# B&R Automation Studio project PallettizerProj_SM
Automation Studio 4.9

## Configuration Config1

### Task classes (Cpu.sw)
```
Cyclic#1:
  SignalHand <- SignalHandler.prg
Cyclic#2:
  Crane <- Crane.prg
  ComTCP_P <- Libraries.ComTCP.ComTCP_P.prg
  Feeder <- Feeder.prg
  InputBridg <- InputBridge.prg
  OutputBrid <- OutputBridge.prg
  PalletHand <- PalletHandler.prg
  MainContro <- MainControl.prg
Cyclic#4:
  InputFilte <- InputFilter.prg
Binaries: udbdef, FWRules, TCData, iomap, ashwac, Role, sysconf, arconfig, asfw, User, ashwd
Libraries: GenericDev, GenericAx, ComTCP_L, operator, standard, AsArLog, AsBrStr, AsTCP, SignalMng, FilterLib, asieccon, astime, runtime
```

### Hardware
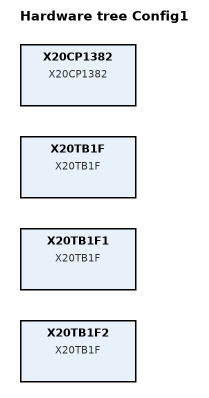
```
X20CP1382 : X20CP1382 v1.14.0.0  [X1 -> X1.SL; X2 -> X2.SL; X3 -> X3.SL]
  Module X1 (Type=X1, Virtual=true, Version=1.14.0.0)
    Connection (Connector=SS1, TargetModule=X20TB1F, TargetConnector=SS)
    Connection (Connector=SL, TargetModule=X20CP1382, TargetConnector=X1)
  Module X2 (Type=X2, Virtual=true, Version=1.14.0.0)
    Connection (Connector=SS1, TargetModule=X20TB1F1, TargetConnector=SS)
    Connection (Connector=SL, TargetModule=X20CP1382, TargetConnector=X2)
  Module X3 (Type=X3, Virtual=true, Version=1.14.0.0)
    Connection (Connector=SS1, TargetModule=X20TB1F2, TargetConnector=SS)
    Connection (Connector=SL, TargetModule=X20CP1382, TargetConnector=X3)
  Connector IF2:
    ActivateDevice = 1
  ConfigurationID = PallettizerProj2_Config1
X20TB1F : X20TB1F v1.0.0.0
X20TB1F1 : X20TB1F v1.0.0.0
X20TB1F2 : X20TB1F v1.0.0.0
```

## Configuration Default_Config

CPU 4PP065.0351-P74, AutomationRuntime C4.72, Build 4.1.2, Vc V4.72.0

### Task classes (Cpu.sw)
```
Cyclic#2:
  ComTCP_P <- Libraries.ComTCP.ComTCP_P.prg
Cyclic#4:
  InputBridg <- InputBridge.prg
  OutputBrid <- OutputBridge.prg
  MainContro <- MainControl.prg
  Feeder <- Feeder.prg
  InputFilte <- InputFilter.prg
Binaries: udbdef, mvLoader, FWRules, TCData, sysconf, Role, User, iomap, ashwd, asfw, arconfig, ashwac, TCLang
Libraries: operator, astime, standard, AsArLog, AsBrStr, AsTCP, runtime, fileio, asieccon, ComTCP_L, GenericDev, GenericAx, FilterLib
```

## Logical view

Binary libraries used (declarations not repeated): operator, runtime, astime, AsIecCon, standard, AsArLog, AsBrStr, AsTCP, MTBasics, brsystem, MTTypes, sys_lib

### Global.var - Global variables
```iecst
(*Constants*)
VAR CONSTANT
	INIT : INT := 0;
	RUN : INT := 1;
END_VAR
VAR
	START_CRANE : BOOL;
	START_PALLET_HANDLER : BOOL;
	START_MACHINE : BOOL;
	START_FEEDER : BOOL;
END_VAR
(*Insert your comment here.*)
VAR
	CraneEnabled : BOOL;
	PalletPositioned : BOOL;
	MoveCrane : BOOL;
	LayerPositioned : BOOL;
	PalletExpultion : BOOL;
	FullPalletReady : BOOL;
	PushLayer : BOOL;
	CraneHomed : BOOL;
END_VAR
(*Sensors*)
VAR
	PALLET_LIGHT_BARRIER_1_IR : BOOL;
	PALLET_LIGHT_BARRIER_2_IR : BOOL;
	LASER_SENSOR_IR : BOOL;
	VACUUM_BOX_CRANE : BOOL;
	LASER_SENSOR_2_IR : BOOL;
	pallet_light_barrier_1 : BOOL;
	pallet_light_barrier_2 : BOOL;
	laser_sensor : BOOL;
	laser_sensor2 : BOOL;
END_VAR
(*Simulation variables*)
VAR
	PUSHER_LBK : BOOL;
	PUSHER_LFR : BOOL;
	TURNPUSHER_LFR : BOOL;
	TURNPUSHER_LBK : BOOL;
	PALLET_FORK_LEFT_FB : BOOL;
	CONVEYOR_IF_FWD : BOOL;
	CONVEYOR_TURN_1_FWD : BOOL;
	PUSHER_FW : BOOL;
	CONVEYOR_END_FWD : BOOL;
	TURNPUSHER_FWD : BOOL;
	TURNPUSHER_BWD : BOOL;
	VACUUM_BOX_CRANE_GRIP : BOOL;
	CARTBOARD_TRIG : BOOL;
	SLIDE_RAIL_RIGHT_EN : BOOL;
	PUSHER_Z_EN : BOOL;
	PUSHER_X_EN : BOOL;
	PALLET_FORK_LEFT_EN : BOOL;
	PALLET_CONVEYOR_1_FWD : BOOL;
	CARRIAGE_2_AXIS : REAL;
	CARRIAGE_2_RCHD : BOOL;
	BOX_CRANE_AXIS : REAL;
	GANTRY_CRANE_AXIS : REAL;
	PALLET_LIFTER_AXIS : REAL;
	BOX_CRANE_TGT_POS : REAL;
	CARRIAGE_2_TGT_POS : REAL;
	GANTRY_CRANE_TGT_POS : REAL;
	PALLET_LIFTER_TGT_POS : REAL;
	PALLET_CONVEYOR_2_ACT_VEL : REAL;
END_VAR
(*Variables*)
VAR
	OperationType : INT := 0;
END_VAR
```

### MNG_Package.var
```iecst
(*                                                                            *)
(* File generated by the B&R AS 4 control config generator                    *)
(*                                                                            *)
(*     Provider: machineering                                                 *)
(*  Application: industrialPhysics_2.4.master                                 *)
(* Architecture: Windows 64 Bit                                               *)
(*      Version: 2.4.10491.master                                             *)
(*        Build: 164f85bec                                                    *)
(*         Date: 2020-05-19, Time: 12:11:21                                   *)
(*                                                                            *)
VAR
	ComTCP_SimInputs : ComTCP_INPUTS_32BIT := (0);
	ComTCP_SimOutputs : ComTCP_OUTPUTS_32BIT := (0);
	ComTCP_SimServerAddress : STRING[15] := '127.0.0.1';
	ComTCP_SimServerPort : UINT := 5000;
	ComTCP_SimSendCycleTime : TIME := T#5ms;
	ComTCP_SimActive : BOOL := FALSE;
END_VAR
(*Signal for the SignalMng*)
VAR
	OnPhaseStopHMI : BOOL;
	AuxReset : BOOL;
	Reset : BOOL;
	ImmediateStopHMI : BOOL;
	NoMorePallet : BOOL;
	OnPhaseStop : BOOL;
	ImmediateStop : BOOL;
	EmergencyStop : BOOL;
	ConveyorIfFault : BOOL;
	ConveyorIfFaultHMI : BOOL;
	ConveyorTurnFault : BOOL;
	ConveyorTurnFaultHMI : BOOL;
	TurnPusherFault : BOOL;
	TurnPusherFaultHMI : BOOL;
	PusherFault : BOOL;
	PusherFaultHMI : BOOL;
	ConveyorEndFault : BOOL;
	ConveyorEndFaultHMI : BOOL;
	CarriageFault : BOOL;
	CarriageFaultHMI : BOOL;
END_VAR
```

### Package Logical/Libraries - Global libraries

### Library Logical/Libraries/GenericDev (IEC)

#### GenericDevice.st
```iecst
(* TODO: Add your comment here *)
FUNCTION_BLOCK GenericDevice

	// Device Clock Handler

	IF (DeviceClock AND (DeviceTimer > 0))THEN
		DeviceTimer := DeviceTimer - 1;
	END_IF;

	// Device Initialization handler

	CASE (DeviceType AND DEVICE_FEEDBACK_MASK) OF

		DEVICE_WITH_ENABLE_FEEDBACK:
			DeviceDisabledSensor := NOT DeviceEnabledSensor AND
			((DeviceState = DeviceDisabledState) OR (DeviceState = DeviceDisablePhaseState AND DeviceTimeout));

			DeviceDisabled := NOT DeviceEnabled AND
			((DeviceState = DeviceDisabledState) OR
			(DeviceState = DeviceDisablePhaseState AND DeviceTimeout));

		DEVICE_WITH_DISABLE_FEEDBACK :
			DeviceEnabled := NOT DeviceDisabled AND
			((DeviceState = DeviceEnabledState) OR
			(DeviceState = DeviceEnablePhaseState AND DeviceTimeout));

			DeviceEnabledSensor := NOT DeviceDisabledSensor AND
			((DeviceState = DeviceEnabledState) OR (DeviceState = DeviceEnablePhaseState AND DeviceTimeout));

		DEVICE_WITHOUT_FEEDBACK:
			DeviceEnabled := (DeviceState = DeviceEnabledState) OR
			(DeviceState = DeviceEnablePhaseState AND DeviceTimeout);
			DeviceDisabled := (DeviceState = DeviceDisabledState) OR
			(DeviceState = DeviceDisablePhaseState AND DeviceTimeout);

			DeviceEnabledSensor := (DeviceState = DeviceEnabledState) OR ((DeviceState = DeviceEnablePhaseState) AND DeviceTimeout);
			DeviceDisabledSensor := (DeviceState = DeviceDisabledState) OR ((DeviceState = DeviceDisablePhaseState) AND DeviceTimeout);
	END_CASE;

	IF (DeviceOperation = INIT) THEN
		// Device sensor handler
		CASE (DeviceType AND DEVICE_FEEDBACK_MASK) OF

			DEVICE_WITH_ENABLE_FEEDBACK:
				DeviceDisabled := NOT DeviceEnabled;

			DEVICE_WITH_DISABLE_FEEDBACK :
				DeviceEnabled := NOT DeviceDisabled;

			DEVICE_WITHOUT_FEEDBACK:
				DeviceEnabled := DeviceEnablePreset;
				DeviceDisabled := NOT DeviceEnabled;
		END_CASE;

		DeviceEnableRequest := FALSE;
		DeviceDisableRequest := FALSE;
		IF (DeviceEnablePreset) THEN
			EnableDevice := TRUE;
			DeviceTimer := DeviceEnableTime;
			IF (NOT (DeviceDisabled AND DeviceEnabled)) THEN
				DeviceState := DeviceEnablePhaseState;
			ELSE
				DeviceState := DeviceEnabledState;
			END_IF;
			DeviceNotInitialized := NOT DeviceEnabled OR DeviceDisabled;
		ELSE
			EnableDevice := FALSE;
			DeviceTimer := DeviceDisableTime;
			IF (NOT (DeviceDisabled AND DeviceEnabled)) THEN
				DeviceState := DeviceDisablePhaseState;
			ELSE
				DeviceState := DeviceDisabledState;
			END_IF;
			DeviceNotInitialized := (DeviceEnabled OR NOT DeviceDisabled);
		END_IF;
	END_IF;

	//	Device control handler

	CASE (DeviceState) OF

		DeviceDisabledState:
			DeviceDisableRequest := FALSE;
			IF (DeviceEnableRequest) THEN
				EnableDevice := TRUE;
				DeviceTimer := DeviceEnableTime;
				DeviceState := DeviceEnablePhaseState;
			END_IF;

		DeviceEnablePhaseState:
			IF DeviceDisableRequest THEN
				DeviceEnableRequest	:= FALSE;
				EnableDevice	:= FALSE;
				DeviceTimer	:= DeviceDisableTime;
				DeviceState	:= DeviceDisablePhaseState;
			END_IF;
			IF DeviceEnabledSensor THEN
				DeviceEnableRequest := FALSE;
				DeviceTimer	:= 0;
				DeviceState := DeviceEnabledState;
			END_IF;

		DeviceEnabledState:
			DeviceEnableRequest	:= FALSE;
			IF DeviceDisableRequest THEN
				EnableDevice := FALSE;
				DeviceTimer	:= DeviceDisableTime;
				DeviceState := DeviceDisablePhaseState;
			END_IF;

		DeviceDisablePhaseState:
			IF DeviceEnableRequest THEN
				DeviceDisableRequest	:= FALSE;
				EnableDevice	:= TRUE;
				DeviceTimer	:= DeviceEnableTime;
				DeviceState	:= DeviceEnablePhaseState;
			END_IF;

			IF DeviceDisabledSensor THEN
				DeviceDisableRequest := FALSE;
				DeviceTimer	:= 0;
				DeviceState := DeviceDisabledState;
			END_IF;

	END_CASE;

	// Device Diagnostic handler

	DeviceTimeout := (DeviceTimer = 0);

	DeviceDisabledSensorFault := ( NOT EnableDevice AND NOT DeviceDisabledSensor AND NOT DeviceEnabledSensor OR EnableDevice AND DeviceDisabledSensor AND DeviceEnabledSensor) AND DeviceTimeout;

	DeviceEnabledSensorFault := (NOT EnableDevice AND DeviceDisabledSensor AND DeviceEnabledSensor OR EnableDevice AND NOT DeviceDisabledSensor AND NOT DeviceEnabledSensor) AND DeviceTimeout;

	DeviceActuatorFault := (NOT EnableDevice AND NOT DeviceDisabledSensor AND DeviceEnabledSensor OR EnableDevice AND DeviceDisabledSensor AND NOT DeviceEnabledSensor) AND DeviceTimeout;

	DeviceFault :=	DeviceDisabledSensorFault OR DeviceEnabledSensorFault OR DeviceActuatorFault;

	// Device actuators handler

	CASE (DeviceType AND DEVICE_ACTUATION_MASK) OF

		DEVICE_WITH_DOUBLE_ACTUATION:
			DisableDevice := NOT EnableDevice;

		DEVICE_WITH_DA_NO_RETAIN:
			EnableDevice := EnableDevice AND (DeviceState = DeviceEnablePhaseState);
			DisableDevice := NOT EnableDevice AND (DeviceState = DeviceDisablePhaseState);

	END_CASE;

END_FUNCTION_BLOCK
```

### Library Logical/Libraries/GenericAx (IEC)

#### Constants.var
```iecst
VAR CONSTANT
	IDLE : WORD := 0;
	CHANGE_VELOCITY : WORD := 1;
	CHANGE_POSITION : WORD := 2;
	IMMEDIATE_STOP_REQUEST : WORD := 3;
	EMERGENCY_STOP_REQUEST : WORD := 4;
END_VAR
```

#### GenericAx.fun
```iecst
FUNCTION_BLOCK GenericAxis
	VAR_INPUT
		Command : WORD := 0;
		ActualPosition : REAL;
		ActualVelocity : REAL;
		NewSetPoint : REAL;
		DeviceTimer : INT;
		TGT_SENSOR : BOOL;
		Reset : BOOL;
	END_VAR
	VAR_OUTPUT
		TargetVelocity : REAL;
		TargetPosition : REAL;
		InPosition : BOOL := 1;
		InVelocity : BOOL := 1;
		DeviceFault : BOOL;
		AxisBusy : BOOL;
	END_VAR
	VAR
		AxisState : GA_State := CheckCommand;
		Timer : INT;
	END_VAR
END_FUNCTION_BLOCK
```

#### GenericAxis.st
```iecst
(* TODO: Add your comment here *)
FUNCTION_BLOCK GenericAxis

	CASE (AxisState) OF

		CheckCommand:

			//			IF Command = IDLE THEN
			//				Timer	:= DeviceTimer;
			//				DeviceFault	:= FALSE;
			//			END_IF;

			IF Command = CHANGE_POSITION THEN

				IF (ActualPosition <> NewSetPoint) THEN
					Timer	:= DeviceTimer;
					InPosition	:= FALSE;
					TargetPosition := NewSetPoint;
					AxisState := WaitTargetPosition;
				END_IF

			END_IF;

			IF Command = CHANGE_VELOCITY THEN

				IF (ActualVelocity <> NewSetPoint) THEN
					Timer	:= DeviceTimer;
					TargetVelocity := NewSetPoint;
					InVelocity	:= FALSE;
					AxisState	:= WaitTargetVelocity;
				END_IF

			END_IF;

//			IF Command = IMMEDIATE_STOP_REQUEST THEN
//
//				TargetPosition	:= ActualPosition;
//				TargetVelocity	:= 0;
//				IF (ActualPosition = TargetPosition AND ActualVelocity = TargetVelocity) THEN
//					InPosition	:= TRUE;
//					InVelocity	:= TRUE;
//					AxisState	:= CheckCommand;
//				END_IF;
//
//			END_IF;

			IF Command = EMERGENCY_STOP_REQUEST THEN
				TargetPosition	:= ActualPosition;
				TargetVelocity	:= 0;
				IF (ActualPosition = TargetPosition AND ActualVelocity = TargetVelocity) THEN
					InPosition	:= TRUE;
					InVelocity	:= TRUE;
					AxisState	:= CheckCommand;
				END_IF;
			END_IF;

		WaitTargetPosition:
			IF (ActualPosition = TargetPosition AND TGT_SENSOR) THEN
				InPosition	:= TRUE;
				AxisState	:= CheckCommand;
			END_IF;
			Timer	:= Timer	- 1;
			IF Timer = 0 THEN
				DeviceFault	:= TRUE;
				AxisState	:= FaultState;
			END_IF;

		WaitTargetVelocity:
			IF ActualVelocity = TargetVelocity THEN
				InVelocity	:= TRUE;
				AxisState	:= CheckCommand;
			END_IF;
			Timer	:= Timer	- 1;
			IF Timer = 0 THEN
				DeviceFault	:= TRUE;
				AxisState	:= FaultState;
			END_IF;

		FaultState:
			IF Reset THEN
				DeviceFault	:= FALSE;
				AxisState	:= CheckCommand;
			END_IF;

	END_CASE;

END_FUNCTION_BLOCK
```

### Library Logical/Libraries/SignalMng (IEC)

#### SignalManagement.st
```iecst
(* TODO: Add your comment here *)
FUNCTION_BLOCK SignalManagement

	CASE SignalOperation OF

		START_CONFIGURATION: (* reset signal count*)

			NumberOfAlarms := 0;
			NumberOfAnomalies := 0;
			NumberOfInformation := 0;
			NumberOfWarnings := 0;

		CONFIGURATION:

			CASE (SignalType AND SIGNAL_TYPE_MASK) OF
				ALARM:
					NumberOfAlarms := NumberOfAlarms + 1;
				ANOMALY:
					NumberOfAnomalies := NumberOfAnomalies + 1;
				WARNING:
					NumberOfWarnings := NumberOfWarnings + 1;
				INFORMATION:
					NumberOfInformation := NumberOfInformation + 1;
			END_CASE

		START_GENERATION:

			ResetEnable := FALSE;
			SignalOutputs := NONE;
			ResetActivation := Reset AND NOT ResetOld;
			ResetOld := Reset;
			AuxResetEnable	:= FALSE;
			AuxResetActivation := KeyReset AND NOT KeyResetOld;
			KeyResetOld:= KeyReset;

		GENERATION:
			CASE (SignalType AND SIGNAL_TYPE_MASK) OF
				ALARM:
					Index := NumberOfActiveAlarms;
					BaseIndex := 0;
					Condition := TRUE;
				ANOMALY:
					Index := NumberOfActiveAnomalies;
					BaseIndex := NumberOfAlarms;
					Condition := TRUE;
				WARNING:
					Index := NumberOfActiveWarning;
					BaseIndex := NumberOfAlarms + NumberOfAnomalies;
					Condition := TRUE;
				INFORMATION:
					Index := NumberOfActiveInformation;
					BaseIndex := NumberOfAlarms + NumberOfAnomalies + NumberOfWarnings;
					Condition := TRUE;
			END_CASE

			IF ActivationSignal AND NOT Signals[SignalCode] THEN
				Signals[SignalCode] := TRUE;
				Index := Index + 1;
				ActiveSignalCodes[BaseIndex + Index] := SignalCode;
			END_IF

			AuxResetRequired := ((SignalType AND AUX_RESET) = AUX_RESET);

			IF (Condition AND Signals[SignalCode] AND NOT ActivationSignal AND (ActiveSignalCodes[BaseIndex + 1] = SignalCode) AND AuxResetRequired) THEN
				AuxResetEnable := TRUE; // LED AUX RECOVERY GREEN
			END_IF

			IF (Condition AND Signals[SignalCode] AND NOT ActivationSignal AND (ActiveSignalCodes[BaseIndex + 1] = SignalCode)) THEN
				ResetEnable := TRUE; // LED RECOVERY GREEN
			END_IF

			IF ((ResetActivation OR NOT Condition) AND Signals[SignalCode] AND NOT ActivationSignal AND (ActiveSignalCodes[BaseIndex + 1] = SignalCode)) THEN
				Signals[SignalCode] := FALSE;

				FOR i := 2 TO Index DO
					ActiveSignalCodes[BaseIndex + i-1] := ActiveSignalCodes[BaseIndex + i];
				END_FOR;

				ActiveSignalCodes[BaseIndex + Index] := 0;
				Index := Index - 1;
				ResetActivation := FALSE;
			END_IF

			IF ((AuxResetActivation OR NOT Condition) AND Signals[SignalCode] AND NOT ActivationSignal AND (ActiveSignalCodes[BaseIndex + 1] = SignalCode) AND AuxResetRequired) THEN
				Signals[SignalCode] := FALSE;

				FOR i := 2 TO Index DO
					ActiveSignalCodes[BaseIndex + i-1] := ActiveSignalCodes[BaseIndex + i];
				END_FOR;

				ActiveSignalCodes[BaseIndex + Index] := 0;
				Index := Index - 1;
				AuxResetActivation := FALSE;
			END_IF

			CASE (SignalType AND SIGNAL_TYPE_MASK) OF
				ALARM:
					NumberOfActiveAlarms := Index;
				ANOMALY:
					NumberOfActiveAnomalies := Index;
				WARNING:
					NumberOfActiveWarning := Index;
				INFORMATION:
					NumberOfActiveInformation := Index;
			END_CASE

			IF Signals[SignalCode] THEN
				SignalOutputs := SignalOutputs OR SignalOutput;
			END_IF

		RUN_SM:
			CurrentAlarm := NumberOfActiveAlarms;
			CurrentAnomaly := NumberOfActiveAnomalies;
			CurrentWarning := NumberOfActiveWarning;
			CurrentInformation := NumberOfActiveInformation;

			IF NumberOfActiveAlarms > 0 THEN
				ActiveAlarmCode := ActiveSignalCodes[CurrentAlarm];
			ELSE
				ActiveAlarmCode := SignalCodeDefault;
			END_IF

			IF NumberOfActiveAnomalies > 0 THEN
				ActiveAnomalyCode := ActiveSignalCodes[NumberOfAlarms + CurrentAnomaly];
			ELSE
				ActiveAnomalyCode := SignalCodeDefault;
			END_IF

			IF NumberOfActiveWarning > 0 THEN
				ActiveWarningCode := ActiveSignalCodes[NumberOfAlarms + NumberOfAnomalies + CurrentWarning];
			ELSE
				ActiveWarningCode := SignalCodeDefault;
			END_IF

			IF NumberOfActiveInformation > 0 THEN
				ActiveInformationCode := ActiveSignalCodes[NumberOfAlarms + NumberOfAnomalies + NumberOfWarnings + CurrentInformation];
			ELSE
				ActiveInformationCode := SignalCodeDefault;
			END_IF;

	END_CASE

END_FUNCTION_BLOCK
```

### Library Logical/Libraries/FilterLib (IEC)

#### FilterLib.fun - Exported functions and function blocks
```iecst
(**)

{REDUND_ERROR} FUNCTION_BLOCK MyFilterFB (*TODO: Add your comment here*) (*$GROUP=User,$CAT=User,$GROUPICON=User.png,$CATICON=User.png*)
	VAR_INPUT
		OperationType : INT;
		Clock : BOOL;
		Signal : BOOL;
		ActivationDelay : UDINT;
		DeactivationDelay : UDINT;
	END_VAR
	VAR_OUTPUT
		DelayedSignal : BOOL;
	END_VAR
	VAR
		Delay : UDINT;
	END_VAR
END_FUNCTION_BLOCK
```

#### MyFilterFB.st
```iecst
(* TODO: Add your comment here *)
FUNCTION_BLOCK MyFilterFB
	IF (OperationType = 0) THEN
		Delay := 0;
	END_IF;
	IF (Clock AND (Delay > 0)) THEN
		Delay := Delay - 1;
	END_IF;
	IF (Delay = 0) THEN
		DelayedSignal := Signal;
	END_IF;
	IF (Signal = DelayedSignal)	THEN
		IF (Signal) THEN
			Delay := DeactivationDelay;
		ELSE
			Delay := ActivationDelay;

		END_IF;
	END_IF;
END_FUNCTION_BLOCK
```

### Program Logical/MainControl (IEC)

#### Main.st
```iecst
PROGRAM _INIT
	(* Insert code here *)

END_PROGRAM

PROGRAM _CYCLIC

	CASE MainState OF

		Initialization:

			IF (OperationType = INIT) THEN

				OperationType := RUN;
				MainState := WaitStart;

			END_IF

		WaitStart:

			IF(START_MACHINE) THEN

				START_FEEDER := TRUE;
				START_CRANE := TRUE;
				START_PALLET_HANDLER := TRUE;
				MainState := WaitCrane;
			END_IF

		WaitCrane:

			IF CraneHomed THEN

				PushLayer := TRUE;
				MainState := WaitFeeder;

			END_IF

			IF FullPalletReady THEN

				PalletExpultion := TRUE;
				MainState := WaitPalletHandler;

			END_IF

		WaitFeeder:

			IF LayerPositioned THEN

				MoveCrane := TRUE;
				MainState := WaitPalletHandler;

			END_IF

		WaitPalletHandler:

			IF OnPhaseStop AND PalletExpultion THEN
				MainState := StopMachine;
			END_IF

			IF PalletPositioned AND NOT (OnPhaseStop AND PalletExpultion) THEN

				CraneEnabled := TRUE;
				MainState := WaitCrane;

			END_IF

		StopMachine:

			START_MACHINE := FALSE;
			START_FEEDER := FALSE;
			START_CRANE := FALSE;
			START_PALLET_HANDLER := FALSE;

			IF Reset THEN

				MainState := WaitStart;

			END_IF

	END_CASE

END_PROGRAM

PROGRAM _EXIT
	(* Insert code here *)

END_PROGRAM
```

### Program Logical/Feeder (IEC)

#### Types.typ
```iecst
TYPE
	FeederStateType :
		(
		WaitStart,
		WaitConv,
		PusherBox,
		BoxCounting,
		BackwardCarriage,
		WaitingBack,
		WaitSyncCrane,
		StopFeederImmediate,
		StopFeederOnPhase,
		WaitingForReactivation
		);
	FeederStruct : 	STRUCT
		State : FeederStateType;
		Start : BOOL;
		Conveyor_if : GenericDevice;
		Conveyor_if_enable_request : BOOL;
		Conveyor_if_disable_request : BOOL;
		Conveyor_if_EnableTime : INT := 20;
		Conveyor_if_DisableTime : INT := 20;
		Conveyor_turn1 : GenericDevice;
		Conveyor_turn1_disable_request : BOOL;
		Conveyor_turn1_enable_request : BOOL;
		Conveyor_turn1_EnableTime : INT := 20;
		Conveyor_turn1_DisableTime : INT := 20;
		Pusher : GenericDevice;
		Pusher_disable_request : BOOL;
		Pusher_enable_request : BOOL;
		PusherEnableTime : INT := 200;
		PusherDisableTime : INT := 200;
		Conveyor_end : GenericDevice;
		Conveyor_end_disable_request : BOOL;
		Conveyor_end_enable_request : BOOL;
		Conveyor_end_EnableTime : INT := 20;
		Conveyor_end_DisableTime : INT := 20;
		Turnpusher : GenericDevice;
		Turnpusher_enable_request : BOOL;
		Turnpusher_disable_request : BOOL;
		TurnpusherEnableTime : INT := 200;
		TurnpusherDisableTime : INT := 200;
		Carriage : GenericAxis;
		CarriagePositionReached : BOOL;
	END_STRUCT;
END_TYPE
```

#### Variables.var
```iecst
VAR
	StopRequest : BOOL := FALSE;
	Box : INT;
	Format : INT := 1;
	Line : INT := 1;
	F_TRIG_0 : F_TRIG;
	LaserSensor2 : BOOL;
	LayerOn : BOOL;
	Feeder : FeederStruct;
	LastLayer : BOOL;
	PrevState : FeederStateType;
	ExpectedBox : INT;
END_VAR
```

#### Main.st
```iecst
PROGRAM _INIT
	(* Insert code here *)

END_PROGRAM

PROGRAM _CYCLIC

	// Falling edge in the coining boxes sensor
	F_TRIG_0( CLK:=LASER_SENSOR_2_IR );
	LaserSensor2 := F_TRIG_0.Q;

	Feeder.Start := START_FEEDER;

	CASE (Feeder.State) OF

		WaitStart:

			IF ImmediateStop THEN

				PrevState := WaitStart;
				Feeder.State := StopFeederImmediate;

			ELSIF Feeder.Start THEN

				Feeder.Conveyor_if_enable_request := TRUE;
				Feeder.Conveyor_turn1_enable_request := TRUE;
				Feeder.Conveyor_end_enable_request := TRUE;

				Feeder.State := WaitConv;

			END_IF

		WaitConv:

			IF ImmediateStop THEN

				Feeder.Conveyor_if_disable_request := TRUE;
				Feeder.Conveyor_end_disable_request := TRUE;
				Feeder.Conveyor_turn1_disable_request := TRUE;

				PrevState := WaitConv;
				Feeder.State := StopFeederImmediate;

			ELSIF NOT Feeder.Conveyor_if_enable_request AND NOT Feeder.Conveyor_turn1_enable_request AND NOT Feeder.Conveyor_end_enable_request THEN

				Feeder.State := PusherBox;

			END_IF

		PusherBox:

			IF ImmediateStop THEN

				Feeder.Conveyor_if_disable_request := TRUE;
				Feeder.Conveyor_end_disable_request := TRUE;
				Feeder.Conveyor_turn1_disable_request := TRUE;

				PrevState := PusherBox;
				Feeder.State := StopFeederImmediate;

			// Behaviour with an OnPhase stop signal
			ELSIF LastLayer AND OnPhaseStop THEN

				Feeder.Conveyor_if_disable_request := TRUE;
				Feeder.Conveyor_end_disable_request := TRUE;
				Feeder.State := StopFeederOnPhase;

			// Nominal behaviour
			ELSIF NOT Feeder.Turnpusher_enable_request AND NOT Feeder.Turnpusher_disable_request AND Feeder.CarriagePositionReached THEN

				IF LASER_SENSOR_IR AND NOT Feeder.Pusher_disable_request THEN
					ExpectedBox := Box + 1;
					Feeder.Pusher_enable_request := TRUE;
					LastLayer := FALSE;
					Feeder.State := BoxCounting;
				END_IF

				IF Box <> ExpectedBox THEN
					Feeder.Pusher_enable_request := TRUE;
					LastLayer := FALSE;
					Feeder.State := BoxCounting;
				END_IF

			END_IF

		BoxCounting:

			IF ImmediateStop THEN

				Feeder.Conveyor_if_disable_request := TRUE;
				Feeder.Conveyor_end_disable_request := TRUE;
				Feeder.Conveyor_turn1_disable_request := TRUE;
				PrevState := BoxCounting;
				Feeder.State := StopFeederImmediate;

			// Nominal
			ELSIF NOT Feeder.Pusher_enable_request THEN

				Feeder.Pusher_disable_request := TRUE;
				LayerPositioned := FALSE;
				LayerOn := FALSE;

				IF LaserSensor2 THEN
					Box := Box+1;

					// Type of boxes in the pallet (first horizzontals)
					IF Format = 1 AND Line = 1 AND Box = 8 THEN
						Feeder.Turnpusher_enable_request := TRUE;
						Line := 2;
						Box := 0;
						ExpectedBox := 0;
						Feeder.Carriage.NewSetPoint	:= 0.44;
						Feeder.Carriage.Command := CHANGE_POSITION;
						Feeder.State := BackwardCarriage;
					END_IF

					IF Format = 1 AND Line = 2 AND Box = 3 THEN
						Line := 3;
						Feeder.Carriage.NewSetPoint	:= 0.44;
						Feeder.Carriage.Command := CHANGE_POSITION;
						Feeder.State := BackwardCarriage;
					END_IF

					IF Format = 1 AND Line = 3 AND Box = 6 THEN
						Line := 1;
						Format := 2;
						Box := 0;
						ExpectedBox := 0;
						Feeder.State := WaitSyncCrane;
					END_IF

					IF Format = 2 AND Line = 1 AND Box = 3 THEN
						Line := 2;
						Feeder.Carriage.NewSetPoint	:= 0.44;
						Feeder.Carriage.Command := CHANGE_POSITION;
						Feeder.State := BackwardCarriage;
					END_IF

					IF Format = 2 AND Line = 2 AND Box = 6 THEN
						Feeder.Turnpusher_disable_request := TRUE;
						Line := 3;
						Box := 0;
						ExpectedBox := 0;
						Feeder.Carriage.NewSetPoint := 0.44;
						Feeder.Carriage.Command := CHANGE_POSITION;
						Feeder.State := BackwardCarriage;
					END_IF

					IF Format = 2 AND Line = 3 AND Box = 8 THEN
						LastLayer := TRUE;
						Line := 1;
						Format := 1;
						Box := 0;
						ExpectedBox := 0;
						Feeder.State := WaitSyncCrane;
					END_IF

					IF (Feeder.State <> BackwardCarriage) AND (Feeder.State <> WaitSyncCrane) THEN
						Feeder.State := PusherBox;
					END_IF
				END_IF

			END_IF

		BackwardCarriage:

			IF ImmediateStop THEN

				Feeder.Conveyor_if_disable_request := TRUE;
				Feeder.Conveyor_end_disable_request := TRUE;
				Feeder.Conveyor_turn1_disable_request := TRUE;

				PrevState := BackwardCarriage;
				Feeder.State := StopFeederImmediate;

			ELSIF Feeder.CarriagePositionReached THEN

				Feeder.Carriage.NewSetPoint := 0.0;
				Feeder.Carriage.Command := CHANGE_POSITION;
				Feeder.State := WaitingBack;

			END_IF

		WaitingBack:

			IF ImmediateStop THEN

				Feeder.Conveyor_if_disable_request := TRUE;
				Feeder.Conveyor_end_disable_request := TRUE;
				Feeder.Conveyor_turn1_disable_request := TRUE;

				PrevState := WaitingBack;
				Feeder.State := StopFeederImmediate;

			ELSIF LayerOn AND Feeder.CarriagePositionReached THEN
				LayerPositioned := TRUE;
				Feeder.State := PusherBox;

			ELSIF NOT LayerOn AND Feeder.CarriagePositionReached THEN
				Feeder.State := PusherBox;
			END_IF

		WaitSyncCrane:

			IF ImmediateStop THEN

				Feeder.Conveyor_if_disable_request := TRUE;
				Feeder.Conveyor_end_disable_request := TRUE;
				Feeder.Conveyor_turn1_disable_request := TRUE;

				PrevState := WaitSyncCrane;
				Feeder.State := StopFeederImmediate;

			ELSIF PushLayer THEN
				Feeder.Carriage.NewSetPoint	:= 1.1;
				Feeder.Carriage.Command := CHANGE_POSITION;
				LayerOn := TRUE;
				PushLayer := FALSE;
				Feeder.State := BackwardCarriage;
			END_IF

		StopFeederImmediate:

			IF LaserSensor2 THEN
				Box := Box+1;
			END_IF

			IF  NOT Feeder.Conveyor_if_disable_request AND NOT Feeder.Conveyor_end_disable_request AND NOT Feeder.Conveyor_turn1_disable_request
				AND NOT ImmediateStop THEN

				Feeder.Conveyor_if_enable_request := TRUE;
				Feeder.Conveyor_end_enable_request := TRUE;
				Feeder.Conveyor_turn1_enable_request := TRUE;
				Feeder.State := WaitingForReactivation;

			END_IF

		StopFeederOnPhase:

			IF NOT Feeder.Conveyor_if_disable_request AND NOT Feeder.Conveyor_end_disable_request AND NOT OnPhaseStop AND NOT ImmediateStop THEN

				Feeder.State := WaitStart;

			END_IF

		WaitingForReactivation:

			IF LaserSensor2 THEN
				Box := Box+1;
			END_IF

			IF NOT Feeder.Conveyor_if_enable_request AND NOT Feeder.Conveyor_end_enable_request AND NOT Feeder.Conveyor_turn1_enable_request THEN

				IF Box <> ExpectedBox THEN
					Feeder.State := BoxCounting;
				END_IF

				IF Box = ExpectedBox THEN
					Feeder.Pusher_disable_request := TRUE;
					Feeder.State := PusherBox;
				END_IF

			END_IF

	END_CASE

	Feeder.Conveyor_if.DeviceOperation := OperationType;
	Feeder.Conveyor_if.DeviceClock := TRUE;
	Feeder.Conveyor_if.DeviceDiagnosticsEnabled := TRUE;
	Feeder.Conveyor_if.DeviceEnablePreset := FALSE;
	Feeder.Conveyor_if.DeviceEnableTime := Feeder.Conveyor_if_EnableTime;
	Feeder.Conveyor_if.DeviceDisableTime := Feeder.Conveyor_if_DisableTime;
	Feeder.Conveyor_if.DeviceType := DEVICE_WITHOUT_FEEDBACK OR DEVICE_WITH_SINGLE_ACTUATION;
	Feeder.Conveyor_if(DeviceEnableRequest := Feeder.Conveyor_if_enable_request, DeviceDisableRequest := Feeder.Conveyor_if_disable_request);
	CONVEYOR_IF_FWD := Feeder.Conveyor_if.EnableDevice;
	ConveyorIfFault	:= Feeder.Conveyor_if.DeviceFault;

	Feeder.Conveyor_turn1.DeviceOperation := OperationType;
	Feeder.Conveyor_turn1.DeviceClock := TRUE;
	Feeder.Conveyor_turn1.DeviceDiagnosticsEnabled := TRUE;
	Feeder.Conveyor_turn1.DeviceEnablePreset := FALSE;
	Feeder.Conveyor_turn1.DeviceEnableTime := Feeder.Conveyor_turn1_EnableTime;
	Feeder.Conveyor_turn1.DeviceDisableTime := Feeder.Conveyor_turn1_DisableTime;
	Feeder.Conveyor_turn1.DeviceType := DEVICE_WITHOUT_FEEDBACK OR DEVICE_WITH_SINGLE_ACTUATION;
	Feeder.Conveyor_turn1(DeviceEnableRequest := Feeder.Conveyor_turn1_enable_request, DeviceDisableRequest := Feeder.Conveyor_turn1_disable_request);
	CONVEYOR_TURN_1_FWD := Feeder.Conveyor_turn1.EnableDevice;
	ConveyorTurnFault := Feeder.Conveyor_turn1.DeviceFault;

	Feeder.Pusher.DeviceOperation := OperationType;
	Feeder.Pusher.DeviceClock := TRUE;
	Feeder.Pusher.DeviceDiagnosticsEnabled := TRUE;
	Feeder.Pusher.DeviceEnablePreset := FALSE;
	Feeder.Pusher.DeviceEnabledSensor := PUSHER_LFR;
	Feeder.Pusher.DeviceDisabledSensor := PUSHER_LBK;
	Feeder.Pusher.DeviceEnableTime := Feeder.PusherEnableTime;
	Feeder.Pusher.DeviceDisableTime := Feeder.PusherDisableTime;
	Feeder.Pusher.DeviceType := DEVICE_WITH_DOUBLE_FEEDBACK OR DEVICE_WITH_SINGLE_ACTUATION;
	Feeder.Pusher(DeviceEnableRequest := Feeder.Pusher_enable_request, DeviceDisableRequest := Feeder.Pusher_disable_request);
	PUSHER_FW := Feeder.Pusher.EnableDevice;
	PusherFault := Feeder.Pusher.DeviceActuatorFault;

	Feeder.Conveyor_end.DeviceOperation := OperationType;
	Feeder.Conveyor_end.DeviceClock := TRUE;
	Feeder.Conveyor_end.DeviceDiagnosticsEnabled := TRUE;
	Feeder.Conveyor_end.DeviceEnablePreset := FALSE;
	Feeder.Conveyor_end.DeviceEnableTime := Feeder.Conveyor_end_EnableTime;
	Feeder.Conveyor_end.DeviceDisableTime := Feeder.Conveyor_end_DisableTime;
	Feeder.Conveyor_end.DeviceType := DEVICE_WITHOUT_FEEDBACK OR DEVICE_WITH_SINGLE_ACTUATION;
	Feeder.Conveyor_end(DeviceEnableRequest := Feeder.Conveyor_end_enable_request, DeviceDisableRequest := Feeder.Conveyor_end_disable_request);
	CONVEYOR_END_FWD := Feeder.Conveyor_end.EnableDevice;
	ConveyorEndFault:= Feeder.Conveyor_end.DeviceFault;

	Feeder.Turnpusher.DeviceOperation := OperationType;
	Feeder.Turnpusher.DeviceClock := TRUE;
	Feeder.Turnpusher.DeviceDiagnosticsEnabled := TRUE;
	Feeder.Turnpusher.DeviceEnablePreset := FALSE;
	Feeder.Turnpusher.DeviceEnabledSensor := TURNPUSHER_LBK;
	Feeder.Turnpusher.DeviceDisabledSensor := TURNPUSHER_LFR;
	Feeder.Turnpusher.DeviceEnableTime := Feeder.TurnpusherEnableTime;
	Feeder.Turnpusher.DeviceDisableTime := Feeder.TurnpusherDisableTime;
	Feeder.Turnpusher.DeviceType := DEVICE_WITH_DOUBLE_FEEDBACK OR DEVICE_WITH_DOUBLE_ACTUATION;
	Feeder.Turnpusher(DeviceEnableRequest := Feeder.Turnpusher_enable_request, DeviceDisableRequest := Feeder.Turnpusher_disable_request);
	TURNPUSHER_BWD := Feeder.Turnpusher.EnableDevice;
	TURNPUSHER_FWD := Feeder.Turnpusher.DisableDevice;
	TurnPusherFault := Feeder.Turnpusher.DeviceActuatorFault;

	Feeder.Carriage.ActualPosition	:= CARRIAGE_2_AXIS;
	CARRIAGE_2_TGT_POS	:= Feeder.Carriage.TargetPosition;
	Feeder.Carriage.TGT_SENSOR	:= CARRIAGE_2_RCHD;
	Feeder.Carriage.DeviceTimer := 400;
	CarriageFault := Feeder.Carriage.DeviceFault;
	Feeder.Carriage();
	Feeder.CarriagePositionReached	:= Feeder.Carriage.InPosition;

END_PROGRAM

PROGRAM _EXIT
	(* Insert code here *)

END_PROGRAM
```

### Program Logical/Crane (IEC)

#### Variables.var
```iecst
VAR
	Crane : CraneStruct;
	NextLayer : INT := 1;
	PrevState : CraneStateType := GoBack;
	CraneState : CraneStateType := 0;
	BoxCraneAxisBusy : BOOL;
	NextState : CraneStateType;
	CompleatingPallet : BOOL;
END_VAR
```

#### Main.st
```iecst
PROGRAM _INIT
	(* Insert code here *)

END_PROGRAM

PROGRAM _CYCLIC

	Crane.Start := START_CRANE;

	CASE (Crane.State) OF

		WaitStart:
			IF Crane.Start THEN
				Crane.State := MoveCraneForCartboard;
			END_IF

		WaitLayer:
			IF Crane.BoxCranePositionReached THEN
				CraneHomed := TRUE;

				IF MoveCrane THEN
					MoveCrane := FALSE;
					Crane.PusherZ_enable_request := TRUE;
					Crane.SlideRail_enable_request := TRUE;
					CraneHomed := FALSE;
					IF (NextLayer = 1) THEN
						Crane.State := ReleaseFirstCartboard;
					END_IF

					IF (NextLayer = 2) THEN
						Crane.State := ReleaseSecondCartboard;
					END_IF
				END_IF
			END_IF

		ReleaseFirstCartboard:

			IF (NOT Crane.PusherZ_enable_request AND NOT Crane.SlideRail_enable_request) AND CraneEnabled THEN

				NextLayer := 2;
				PrevState := ReleaseFirstCartboard;
				Crane.GantryCrane.NewSetPoint := -1.11;
				Crane.GantryCrane.Command := CHANGE_POSITION;
				Crane.BoxCrane.NewSetPoint := -0.2;
				Crane.BoxCrane.Command := CHANGE_POSITION;
				Crane.State := WaitingPositioning;

			END_IF

		PositioningLayer:

			IF NOT Crane.Vacuum_disable_request AND NOT VACUUM_BOX_CRANE THEN

				PrevState := PositioningLayer;
				Crane.GantryCrane.NewSetPoint := -1.3;
				Crane.GantryCrane.Command := CHANGE_POSITION;
				Crane.State := WaitingPositioning;

			END_IF

		LayerOnPallet:

			IF NOT Crane.SlideRail_disable_request THEN

				Crane.PusherX_enable_request := TRUE ;
				Crane.GantryCrane.NewSetPoint := 0.0;
				Crane.GantryCrane.Command := CHANGE_POSITION;
				PrevState := LayerOnPallet;
				Crane.State := WaitingPositioning;

			END_IF

		GoBack:

			IF FullPalletReady AND OnPhaseStop THEN

				Crane.PusherZ_disable_request := TRUE;
				Crane.PusherX_disable_request := TRUE;
				Crane.BoxCrane.NewSetPoint := 0.0;
				Crane.BoxCrane.Command := CHANGE_POSITION;
				NextState := StopCrane;
				PrevState := GoBack;
				Crane.State := WaitingPositioning;

			END_IF

			CraneEnabled := FALSE;
			FullPalletReady := FALSE;

			IF PrevState = LayerOnPallet AND NOT Crane.PusherX_enable_request THEN

				Crane.PusherZ_disable_request := TRUE;
				Crane.PusherX_disable_request := TRUE;
				Crane.BoxCrane.NewSetPoint := 0.0;
				Crane.BoxCrane.Command := CHANGE_POSITION;
				NextState := MoveCraneForCartboard;
				PrevState := GoBack;
				Crane.State := WaitingPositioning;

			END_IF

			IF (PrevState = LoadCartboard AND NOT Crane.Vacuum_enable_request) THEN

				Crane.BoxCrane.NewSetPoint := 0.0;
				Crane.BoxCrane.Command := CHANGE_POSITION;
				NextState := WaitLayer;
				PrevState := GoBack;
				Crane.State := WaitingPositioning;

			END_IF

		MoveCraneForCartboard:

			IF Crane.BoxCranePositionReached THEN

				Crane.BoxCrane.NewSetPoint := -0.195;
				Crane.BoxCrane.Command := CHANGE_POSITION;
				Crane.State := LoadCartboard;

			END_IF

		LoadCartboard:

			IF Crane.BoxCranePositionReached THEN

				Crane.Vacuum_enable_request	:= TRUE;
				Crane.Cartboard_enable_request := TRUE;
				PrevState := LoadCartboard;
				Crane.State := GoBack;

			END_IF

		ReleaseSecondCartboard:

			IF (NOT Crane.PusherZ_enable_request AND NOT Crane.SlideRail_enable_request) THEN

				NextLayer := 1;
				Crane.GantryCrane.NewSetPoint := -1.11;
				Crane.GantryCrane.Command := CHANGE_POSITION;
				Crane.BoxCrane.NewSetPoint := 0.01;
				Crane.BoxCrane.Command := CHANGE_POSITION;
				CompleatingPallet := TRUE;
				PrevState := ReleaseSecondCartboard;
				Crane.State := WaitingPositioning;

			END_IF

		WaitingPositioning:

			IF Crane.GantryCranePositionReached AND Crane.BoxCranePositionReached    (*GANTRY_CRANE_AXIS = -1.11 AND BOX_CRANE_AXIS = 0.01*) THEN

				IF PrevState = ReleaseFirstCartboard OR PrevState = ReleaseSecondCartboard THEN

					Crane.Vacuum_disable_request := TRUE;
					Crane.Cartboard_disable_request := TRUE;
					Crane.State := PositioningLayer;

				END_IF

				IF PrevState = PositioningLayer THEN

					Crane.SlideRail_disable_request := TRUE;
					Crane.State := LayerOnPallet;

				END_IF

				IF PrevState = LayerOnPallet THEN

					IF CompleatingPallet THEN
						CompleatingPallet:=FALSE;
						FullPalletReady := TRUE;
					END_IF

					Crane.State := GoBack;

				END_IF

				IF PrevState = GoBack THEN

					Crane.State := NextState;

				END_IF

			END_IF

		StopCrane:

			IF Reset THEN

				Crane.State := WaitStart;

			END_IF

	END_CASE

	Crane.Vacuum.DeviceOperation := OperationType;
	Crane.Vacuum.DeviceClock := TRUE;
	Crane.Vacuum.DeviceDiagnosticsEnabled := TRUE;
	Crane.Vacuum.DeviceEnablePreset := FALSE;
	Crane.Vacuum.DeviceEnabledSensor := VACUUM_BOX_CRANE;
	Crane.Vacuum.DeviceEnableTime := 500;//VacuumEnableTime;
	Crane.Vacuum.DeviceDisableTime := Crane.VacuumDisableTime;
	Crane.Vacuum.DeviceType := DEVICE_WITH_SINGLE_ACTUATION OR DEVICE_WITH_ENABLE_FEEDBACK;
	Crane.Vacuum(DeviceEnableRequest := Crane.Vacuum_enable_request, DeviceDisableRequest := Crane.Vacuum_disable_request );
	VACUUM_BOX_CRANE_GRIP := Crane.Vacuum.EnableDevice;
	//eVacuumFault := (*Vacuum.DeviceEnabledSensorFault OR Vacuum.DeviceActuatorFault*) SIMVacuumFault;

	Crane.Cartboard.DeviceOperation := OperationType;
	Crane.Cartboard.DeviceClock := TRUE;
	Crane.Cartboard.DeviceDiagnosticsEnabled := TRUE;
	Crane.Cartboard.DeviceEnablePreset := FALSE;
	Crane.Cartboard.DeviceEnableTime := Crane.CartboardEnableTime;
	Crane.Cartboard.DeviceDisableTime := Crane.CartboardDisableTime;
	Crane.Cartboard.DeviceType := DEVICE_WITHOUT_FEEDBACK OR DEVICE_WITH_SINGLE_ACTUATION;
	Crane.Cartboard(DeviceEnableRequest := Crane.Cartboard_enable_request, DeviceDisableRequest := Crane.Cartboard_disable_request);
	CARTBOARD_TRIG := Crane.Cartboard.EnableDevice;
//	eCartboardFault	:= (*Cartboard.DeviceActuatorFault*) SIMCartboardFault;

	Crane.SlideRail.DeviceOperation := OperationType;
	Crane.SlideRail.DeviceClock := TRUE;
	Crane.SlideRail.DeviceDiagnosticsEnabled := TRUE;
	Crane.SlideRail.DeviceEnablePreset := FALSE;
	Crane.SlideRail.DeviceEnableTime := Crane.SlideRailEnableTime;
	Crane.SlideRail.DeviceDisableTime := Crane.SlideRailDisableTime;
	Crane.SlideRail.DeviceType := DEVICE_WITHOUT_FEEDBACK OR DEVICE_WITH_SINGLE_ACTUATION;
	Crane.SlideRail(DeviceEnableRequest := Crane.SlideRail_enable_request, DeviceDisableRequest := Crane.SlideRail_disable_request);
	SLIDE_RAIL_RIGHT_EN := Crane.SlideRail.EnableDevice;
	//eSlideRailFault	:= (*SlideRail.DeviceActuatorFault*) SIMSlideRailFault;

	Crane.PusherZ.DeviceOperation := OperationType;
	Crane.PusherZ.DeviceClock := TRUE;
	Crane.PusherZ.DeviceDiagnosticsEnabled := TRUE;
	Crane.PusherZ.DeviceEnablePreset := FALSE;
	Crane.PusherZ.DeviceEnableTime := Crane.PusherZEnableTime;
	Crane.PusherZ.DeviceDisableTime := Crane.PusherZDisableTime;
	Crane.PusherZ.DeviceType := DEVICE_WITHOUT_FEEDBACK OR DEVICE_WITH_SINGLE_ACTUATION;
	Crane.PusherZ(DeviceEnableRequest := Crane.PusherZ_enable_request, DeviceDisableRequest := Crane.PusherZ_disable_request);
	PUSHER_Z_EN := Crane.PusherZ.EnableDevice;
	//ePusherzFault	:= (*PusherZ.DeviceActuatorFault*) SIMPusherzFault;

	Crane.PusherX.DeviceOperation := OperationType;
	Crane.PusherX.DeviceClock := TRUE;
	Crane.PusherX.DeviceDiagnosticsEnabled := TRUE;
	Crane.PusherX.DeviceEnablePreset := FALSE;
	Crane.PusherX.DeviceEnableTime := Crane.PusherXEnableTime;
	Crane.PusherX.DeviceDisableTime := Crane.PusherXDisableTime;
	Crane.PusherX.DeviceType := DEVICE_WITHOUT_FEEDBACK OR DEVICE_WITH_SINGLE_ACTUATION;
	Crane.PusherX(DeviceEnableRequest := Crane.PusherX_enable_request, DeviceDisableRequest := Crane.PusherX_disable_request );
	PUSHER_X_EN := Crane.PusherX.EnableDevice;
	//ePusherxFault	:= (*PusherX.DeviceActuatorFault*) SIMPusherxFault;

	Crane.GantryCrane.ActualPosition	:= GANTRY_CRANE_AXIS;
	Crane.GantryCrane.TGT_SENSOR	:= TRUE;
	GANTRY_CRANE_TGT_POS	:= Crane.GantryCrane.TargetPosition;
	Crane.GantryCrane.DeviceTimer	:= 400;
	//eGantryCraneFault	:= (*GantryCrane.DeviceFault*) SIMGantryCraneFault;
	Crane.GantryCrane();
	Crane.GantryCranePositionReached	:= Crane.GantryCrane.InPosition;

	//BoxCrane.NewSetPoint	:= BoxCraneSetPoint;
	Crane.BoxCrane.ActualPosition	:= BOX_CRANE_AXIS;
	Crane.BoxCrane.TGT_SENSOR	:= TRUE;
	BOX_CRANE_TGT_POS	:=	Crane.BoxCrane.TargetPosition;
	Crane.BoxCrane.DeviceTimer	:= 400;
	//eBoxCraneFault	:= (*BoxCrane.DeviceFault*) SIMBoxCraneFault;
	Crane.BoxCrane();
	Crane.BoxCranePositionReached	:= Crane.BoxCrane.InPosition;

END_PROGRAM

PROGRAM _EXIT
	(* Insert code here *)

END_PROGRAM
```

### Program Logical/PalletHandler (IEC)

#### Types.typ
```iecst
TYPE
	PalletStruct : 	STRUCT
		Start : BOOL;
		State : PalletStateType;
		PalletFork : GenericDevice;
		PalletFork_enable_request : BOOL;
		PalletFork_disable_request : BOOL;
		PalletForkEnableTime : INT := 20;
		PalletForkDisableTime : INT := 20;
		PalletLifter : GenericAxis;
		PalletLifterPositionReached : BOOL;
		PalletConveyor1 : GenericDevice;
		PalletConveyor1EnableTime : INT := 20;
		PalletConveyor1DisableTime : INT := 20;
		PalletConveyor2 : GenericAxis;
		PalletConveyor1_disable_request : BOOL;
		PalletConveyor1_enable_request : BOOL;
		PalletConveyor2VelocityReached : BOOL;
	END_STRUCT;
	PalletStateType :
		(
		WaitStart,
		ReleasePallet,
		NextPallet,
		LifterHoming,
		MovingPallet,
		PositioningPallet,
		PalletApproaching,
		PalletInPosition,
		WaitingPositioning,
		StopPalletOnPhase,
		StopPalletImmediate
		);
END_TYPE
```

#### Main.st
```iecst
PROGRAM _INIT

	NumberPallet := 5;

END_PROGRAM

PROGRAM _CYCLIC

	Pallet.Start := START_PALLET_HANDLER;

	CASE (Pallet.State) OF

		WaitStart:

			IF ImmediateStop THEN

				PrevState := WaitStart;
				Pallet.State := StopPalletImmediate;

			ELSIF Pallet.Start THEN
				Pallet.State := ReleasePallet;
			END_IF

		ReleasePallet:

			PalletExpultion := FALSE;
			PalletPositioned := FALSE;

			IF ImmediateStop THEN

				Pallet.PalletConveyor2.NewSetPoint := 0.0;
				Pallet.PalletConveyor2.Command := CHANGE_VELOCITY;

				PrevState := ReleasePallet;
				Pallet.State :=StopPalletImmediate;

			ELSIF Pallet.PalletLifterPositionReached AND NOT OnPhaseStop THEN

				Pallet.PalletConveyor2.NewSetPoint := 0.5;
				Pallet.PalletConveyor2.Command := CHANGE_VELOCITY;
				Pallet.PalletLifter.NewSetPoint := -0.258;
				Pallet.PalletLifter.Command := CHANGE_POSITION;

				PrevState := ReleasePallet;
				Pallet.State := WaitingPositioning;

			END_IF

		NextPallet:

			IF ImmediateStop THEN

				Pallet.PalletConveyor2.NewSetPoint := 0.0;
				Pallet.PalletConveyor2.Command := CHANGE_VELOCITY;

				PrevState := NextPallet;
				Pallet.State :=StopPalletImmediate;

			ELSIF NOT Pallet.PalletFork_enable_request THEN

				Pallet.PalletLifter.NewSetPoint := -0.12;
				Pallet.PalletLifter.Command := CHANGE_POSITION;

				PrevState := NextPallet;
				Pallet.State := WaitingPositioning;

			END_IF

		LifterHoming:

			IF ImmediateStop THEN

				Pallet.PalletConveyor2.NewSetPoint := 0.0;
				Pallet.PalletConveyor2.Command := CHANGE_VELOCITY;

				PrevState := LifterHoming;
				Pallet.State :=StopPalletImmediate;

			ELSIF NOT Pallet.PalletFork_disable_request THEN
				Pallet.PalletLifter.NewSetPoint := 0.0;
				Pallet.PalletLifter.Command := CHANGE_POSITION;

				Pallet.State := MovingPallet;
			END_IF

		MovingPallet:

			IF ImmediateStop THEN

				Pallet.PalletConveyor2.NewSetPoint := 0.0;
				Pallet.PalletConveyor2.Command := CHANGE_VELOCITY;

				PrevState := MovingPallet;
				Pallet.State :=StopPalletImmediate;

			ELSIF Pallet.PalletLifterPositionReached THEN

				Pallet.PalletConveyor1_enable_request := TRUE;
				Pallet.PalletLifter.NewSetPoint := 0.0;
				Pallet.PalletLifter.Command := CHANGE_POSITION;
				Pallet.State := PositioningPallet;

			END_IF

		PositioningPallet:

			IF ImmediateStop THEN

				Pallet.PalletConveyor2.NewSetPoint := 0.0;
				Pallet.PalletConveyor2.Command := CHANGE_VELOCITY;
				Pallet.PalletConveyor1_disable_request := TRUE;

				PrevState := PositioningPallet;
				Pallet.State :=StopPalletImmediate;

			ELSIF Pallet.PalletConveyor2VelocityReached AND NOT Pallet.PalletConveyor1_enable_request AND PALLET_LIGHT_BARRIER_2_IR THEN

				Pallet.PalletConveyor2.NewSetPoint := 0.1;
				Pallet.PalletConveyor2.Command := CHANGE_VELOCITY;
				Pallet.State := PalletApproaching;

			END_IF

		PalletApproaching:

			IF ImmediateStop THEN

				Pallet.PalletConveyor2.NewSetPoint := 0.0;
				Pallet.PalletConveyor2.Command := CHANGE_VELOCITY;
				Pallet.PalletConveyor1_disable_request := TRUE;

				PrevState := PalletApproaching;
				Pallet.State :=StopPalletImmediate;

			ELSIF Pallet.PalletConveyor2VelocityReached AND PALLET_LIGHT_BARRIER_1_IR THEN

				Pallet.PalletConveyor2.NewSetPoint := 0.0;
				Pallet.PalletConveyor2.Command := CHANGE_VELOCITY;
				Pallet.PalletConveyor1_disable_request := TRUE;
				Pallet.State := PalletInPosition;

			END_IF

		PalletInPosition:

			IF ImmediateStop THEN

				PrevState := PalletApproaching;
				Pallet.State :=StopPalletImmediate;

			ELSIF Pallet.PalletConveyor2VelocityReached AND NOT Pallet.PalletConveyor1_disable_request THEN

				PalletPositioned := TRUE;

				IF PalletExpultion THEN

					IF OnPhaseStop THEN

						Pallet.PalletConveyor1_disable_request := TRUE;
						Pallet.PalletConveyor2.NewSetPoint := 0.0;
						Pallet.PalletConveyor2.Command := CHANGE_VELOCITY;
						Pallet.State := StopPalletOnPhase;

					END_IF

					IF NOT OnPhaseStop THEN

						Pallet.PalletConveyor2.NewSetPoint := 0.5;
						Pallet.PalletConveyor2.Command := CHANGE_VELOCITY;
						Pallet.State := ReleasePallet;

					END_IF

				END_IF

			END_IF

		WaitingPositioning:

			IF ImmediateStop THEN

				Pallet.PalletConveyor2.NewSetPoint := 0.0;
				Pallet.PalletConveyor2.Command := CHANGE_VELOCITY;
				Pallet.State := StopPalletImmediate;

			ELSIF Pallet.PalletLifterPositionReached THEN

				IF PrevState = ReleasePallet THEN
					NumberPallet := NumberPallet-1;

					IF NumberPallet = 0 THEN
						NoMorePallet := TRUE;
					END_IF

					Pallet.PalletFork_enable_request := TRUE;
					Pallet.State := NextPallet;

				END_IF

				IF PrevState = NextPallet THEN

					Pallet.PalletFork_disable_request := TRUE;
					Pallet.State := LifterHoming;

				END_IF

			END_IF

		StopPalletOnPhase:

			IF NOT Pallet.PalletConveyor1_disable_request AND Pallet.PalletConveyor2VelocityReached  AND NOT OnPhaseStop THEN

				IF NumberPallet = 0 THEN
					NoMorePallet := FALSE;
					NumberPallet := 5;
				END_IF

				Pallet.State := WaitStart;

			END_IF

		StopPalletImmediate:

			IF Pallet.PalletConveyor2VelocityReached AND NOT ImmediateStop THEN

				IF (PrevState = PositioningPallet ) AND NOT Pallet.PalletConveyor1_disable_request THEN

					Pallet.PalletConveyor1_enable_request := TRUE;
					Pallet.PalletConveyor2.NewSetPoint := 0.5;
					Pallet.PalletConveyor2.Command := CHANGE_VELOCITY;

				END_IF

				IF PrevState = PalletApproaching AND NOT Pallet.PalletConveyor1_disable_request THEN

					Pallet.PalletConveyor1_enable_request := TRUE;
					Pallet.PalletConveyor2.NewSetPoint := 0.1;
					Pallet.PalletConveyor2.Command := CHANGE_VELOCITY;

				END_IF

				Pallet.State := PrevState;

			END_IF

	END_CASE

	Pallet.PalletFork.DeviceOperation := OperationType;
	Pallet.PalletFork.DeviceClock := TRUE;
	Pallet.PalletFork.DeviceDiagnosticsEnabled := TRUE;
	Pallet.PalletFork.DeviceEnablePreset := FALSE;
	Pallet.PalletFork.DeviceEnabledSensor := PALLET_FORK_LEFT_FB;
	Pallet.PalletFork.DeviceEnableTime := Pallet.PalletForkEnableTime;
	Pallet.PalletFork.DeviceDisableTime := Pallet.PalletForkDisableTime;
	PALLET_FORK_LEFT_EN := Pallet.PalletFork.EnableDevice;
	Pallet.PalletFork.DeviceType := DEVICE_WITH_ENABLE_FEEDBACK OR DEVICE_WITH_SINGLE_ACTUATION;
	Pallet.PalletFork(DeviceEnableRequest := Pallet.PalletFork_enable_request, DeviceDisableRequest := Pallet.PalletFork_disable_request);
	PalletforkFault := Pallet.PalletFork.DeviceFault;

	Pallet.PalletConveyor1.DeviceOperation := OperationType;
	Pallet.PalletConveyor1.DeviceClock := TRUE;
	Pallet.PalletConveyor1.DeviceDiagnosticsEnabled := TRUE;
	Pallet.PalletConveyor1.DeviceEnablePreset := FALSE;
	Pallet.PalletConveyor1.DeviceEnableTime := Pallet.PalletConveyor1EnableTime;
	Pallet.PalletConveyor1.DeviceDisableTime := Pallet.PalletConveyor1DisableTime;
	Pallet.PalletConveyor1.DeviceType := DEVICE_WITHOUT_FEEDBACK OR DEVICE_WITH_SINGLE_ACTUATION;
	PALLET_CONVEYOR_1_FWD := Pallet.PalletConveyor1.EnableDevice;
	Pallet.PalletConveyor1(DeviceEnableRequest := Pallet.PalletConveyor1_enable_request, DeviceDisableRequest := Pallet.PalletConveyor1_disable_request);
	PalletConveyor1Fault := Pallet.PalletConveyor1.DeviceFault;

	Pallet.PalletLifter.ActualPosition	:= PALLET_LIFTER_AXIS;
	Pallet.PalletLifter.TGT_SENSOR	:= TRUE;
	PALLET_LIFTER_TGT_POS 	:= Pallet.PalletLifter.TargetPosition;
	Pallet.PalletLifter.DeviceTimer	:= 400;
	PalletLifterFault	:= Pallet.PalletLifter.DeviceFault;
	Pallet.PalletLifter();
	Pallet.PalletLifterPositionReached	:= Pallet.PalletLifter.InPosition;

	Pallet.PalletConveyor2.ActualVelocity	:= PALLET_CONVEYOR_2_ACT_VEL;
	PALLET_CONVEYOR_2_ACT_VEL	:= Pallet.PalletConveyor2.TargetVelocity;
	Pallet.PalletConveyor2.DeviceTimer	:= 400;
	PalletConveyor2Fault:= Pallet.PalletConveyor2.DeviceFault;
	Pallet.PalletConveyor2();
	Pallet.PalletConveyor2VelocityReached	:= Pallet.PalletConveyor2.InVelocity;

END_PROGRAM

PROGRAM _EXIT
	(* Insert code here *)

END_PROGRAM
```

### Program Logical/SignalHandler (IEC)

#### Main.st
```iecst
PROGRAM _INIT
	(* Insert code here *)

END_PROGRAM

PROGRAM _CYCLIC

	// Recognize input

	IF (OperationType = INIT) THEN
		SignalManager(SignalOperation := START_CONFIGURATION);
		SignalManager.SignalOperation  := CONFIGURATION;
	ELSE
		SignalManager(SignalOperation 	:= START_GENERATION);
		SignalManager.SignalOperation 	:= GENERATION;
	END_IF;

	SignalManager.ActivationSignal := OnPhaseStopHMI;
	SignalManager.SignalCode := 1;
	SignalManager.SignalType := ANOMALY;
	SignalManager.SignalOutput := ON_PHASE_STOP;
	SignalManager.Reset := Reset;
	SignalManager();

	SignalManager.ActivationSignal := NoMorePallet;
	SignalManager.SignalCode := 2;
	SignalManager.SignalType := ANOMALY;
	SignalManager.SignalOutput := ON_PHASE_STOP;
	SignalManager.Reset := Reset;
	SignalManager();

	SignalManager.ActivationSignal := ImmediateStopHMI;
	SignalManager.SignalCode := 3;
	SignalManager.SignalType := ALARM OR AUX_RESET;
	SignalManager.SignalOutput := IMMEDIATE_STOP;
	SignalManager.KeyReset := AuxReset;
	SignalManager();

	//Feeder
	SignalManager.ActivationSignal :=  ConveyorIfFaultHMI;
	SignalManager.SignalCode := 4;
	SignalManager.SignalType := ALARM OR AUX_RESET;
	SignalManager.SignalOutput := IMMEDIATE_STOP;
	SignalManager.KeyReset := AuxReset;
	SignalManager();

	SignalManager.ActivationSignal := ConveyorEndFaultHMI;
	SignalManager.SignalCode := 5;
	SignalManager.SignalType := ALARM OR AUX_RESET;
	SignalManager.SignalOutput := IMMEDIATE_STOP;
	SignalManager.KeyReset := AuxReset;
	SignalManager();

	SignalManager.ActivationSignal := ConveyorTurnFaultHMI;
	SignalManager.SignalCode := 6;
	SignalManager.SignalType := ALARM OR AUX_RESET;
	SignalManager.SignalOutput := IMMEDIATE_STOP;
	SignalManager.KeyReset := AuxReset;
	SignalManager();

	SignalManager.ActivationSignal := PusherFaultHMI;
	SignalManager.SignalCode := 7;
	SignalManager.SignalType := ALARM OR AUX_RESET;
	SignalManager.SignalOutput := IMMEDIATE_STOP;
	SignalManager.KeyReset := AuxReset;
	SignalManager();

	SignalManager.ActivationSignal := TurnPusherFaultHMI;
	SignalManager.SignalCode := 8;
	SignalManager.SignalType := ALARM OR AUX_RESET;
	SignalManager.SignalOutput := IMMEDIATE_STOP;
	SignalManager.KeyReset := AuxReset;
	SignalManager();

	SignalManager.ActivationSignal := CarriageFaultHMI;
	SignalManager.SignalCode := 9;
	SignalManager.SignalType := ALARM OR AUX_RESET;
	SignalManager.SignalOutput := IMMEDIATE_STOP;
	SignalManager.KeyReset := AuxReset;
	SignalManager();

	EmergencyStop	:= ((SignalManager.SignalOutputs AND EMERGENCY_STOP) = EMERGENCY_STOP);
	ImmediateStop	:= ((SignalManager.SignalOutputs AND IMMEDIATE_STOP) = IMMEDIATE_STOP);
	OnPhaseStop		:= ((SignalManager.SignalOutputs AND ON_PHASE_STOP)  = ON_PHASE_STOP);

END_PROGRAM

PROGRAM _EXIT
	(* Insert code here *)

END_PROGRAM
```

### Program Logical/InputFilter (IEC)

#### Variables.var
```iecst
VAR
	LaserSensor : MyFilterFB;
	LaserSensor2 : MyFilterFB;
	PalletLightBarrierSensor1 : MyFilterFB;
	PalletLightBarrierSensor2 : MyFilterFB;
END_VAR
```

#### Main.st
```iecst
PROGRAM _INIT
	(* Insert code here *)

END_PROGRAM

PROGRAM _CYCLIC

	//Pallet_light_barrier1 filtering
	PalletLightBarrierSensor1.OperationType := OperationType;
	PalletLightBarrierSensor1.Clock := TRUE;
	PalletLightBarrierSensor1.Signal  := PALLET_LIGHT_BARRIER_1_IR;
	PalletLightBarrierSensor1.ActivationDelay := 2;
	PalletLightBarrierSensor1.DeactivationDelay  := 0;
	PalletLightBarrierSensor1();

	pallet_light_barrier_1 := PalletLightBarrierSensor1.DelayedSignal;

	//Pallet_light_barrier2 filtering
	PalletLightBarrierSensor2.OperationType := OperationType;
	PalletLightBarrierSensor2.Clock := TRUE;
	PalletLightBarrierSensor2.Signal  := PALLET_LIGHT_BARRIER_2_IR;
	PalletLightBarrierSensor2.ActivationDelay := 2;
	PalletLightBarrierSensor2.DeactivationDelay  := 0;
	PalletLightBarrierSensor2();

	pallet_light_barrier_2 := PalletLightBarrierSensor2.DelayedSignal;

	//Sensor1 filtering
	LaserSensor.OperationType := OperationType;
	LaserSensor.Clock := TRUE;
	LaserSensor.Signal  := LASER_SENSOR_IR;
	LaserSensor.ActivationDelay := 2;
	LaserSensor.DeactivationDelay  := 0;
	LaserSensor();

	laser_sensor := LaserSensor.DelayedSignal;

	//Sensor2 filtering
	LaserSensor2.OperationType := OperationType;
	LaserSensor2.Clock := TRUE;
	LaserSensor2.Signal  := LASER_SENSOR_2_IR;
	LaserSensor2.ActivationDelay := 2;
	LaserSensor2.DeactivationDelay  := 0;
	LaserSensor2();

	laser_sensor2 := LaserSensor2.DelayedSignal;

END_PROGRAM

PROGRAM _EXIT
	(* Insert code here *)

END_PROGRAM
```

Listed in the project but not available here: Logical/Global.typ, Logical/MNG_Global.typ, Logical/MNG_Package.typ, Logical/Libraries/ComTCP, Logical/Libraries/GenericDev/Types.typ, Logical/Libraries/GenericDev/Constants.var, Logical/Libraries/GenericDev/GenericDev.fun, Logical/Libraries/FilterLib/Types.typ, Logical/Libraries/FilterLib/Constants.var, Logical/InputBridge, Logical/OutputBridge
